ABB RAPID module: ReplayTargets_v22.mod

MODULE ReplayTargets_v22
    ! Generated from tests_v22.csv and success_v22.csv.
    ! Target names include version and testId. B* variants include version, testId, and confId.

    ! Robtargets and jointtargets for replay
    CONST robtarget rA_v22_t1 := [[2085.37,-90.629,2712.24],[0.500386,0.301254,-0.151089,0.797516],[-1,2,3,0],[9E+09,9E+09,9E+09,9E+09,9E+09,9E+09]];
    CONST robtarget rB_v22_t1 := [[2086.58,-104.628,2712.84],[0.500947,0.305697,-0.157375,0.794251],[-1,2,3,0],[9E+09,9E+09,9E+09,9E+09,9E+09,9E+09]];
    CONST robtarget rB_v22_t1_c9 := [[2086.58,-104.628,2712.84],[0.500947,0.305697,-0.157375,0.794251],[0,4,4,0],[9E+09,9E+09,9E+09,9E+09,9E+09,9E+09]];
    CONST jointtarget jA_v22_t1 := [[-0.000990208,21.9,-48.6,225.001,50.1,270.001],[9E+09,9E+09,9E+09,9E+09,9E+09,9E+09]];
    CONST jointtarget jB_v22_t1 := [[-0.330828,22.1227,-48.9906,226.207,50.1732,269.29],[9E+09,9E+09,9E+09,9E+09,9E+09,9E+09]];
    CONST jointtarget jBseed_v22_t1 := [[0,21.9,-48.6,225,50.1,270],[9E+09,9E+09,9E+09,9E+09,9E+09,9E+09]];
    CONST num seedB_v22_t1 := 12121;

    CONST robtarget rA_v22_t2 := [[2569.13,0.0397207,799.136],[0.45399,-6.87952E-6,0.891007,3.17843E-6],[0,-1,4,0],[9E+09,9E+09,9E+09,9E+09,9E+09,9E+09]];
    CONST robtarget rB_v22_t2 := [[2573.15,0.509089,797.884],[0.45376,0.0013057,0.891089,0.00778675],[0,-1,4,0],[9E+09,9E+09,9E+09,9E+09,9E+09,9E+09]];
    CONST robtarget rB_v22_t2_c8 := [[2573.15,0.509089,797.884],[0.45376,0.0013057,0.891089,0.00778675],[0,0,4,0],[9E+09,9E+09,9E+09,9E+09,9E+09,9E+09]];
    CONST jointtarget jA_v22_t2 := [[0.000888186,38.4,-6.4,-0.000518049,4,360],[9E+09,9E+09,9E+09,9E+09,9E+09,9E+09]];
    CONST jointtarget jB_v22_t2 := [[-0.0378482,38.6214,-6.68159,10.5195,4.15455,350.024],[9E+09,9E+09,9E+09,9E+09,9E+09,9E+09]];
    CONST jointtarget jBseed_v22_t2 := [[0,38.4,-6.4,0,4,360],[9E+09,9E+09,9E+09,9E+09,9E+09,9E+09]];
    CONST num seedB_v22_t2 := 701;

    CONST robtarget rA_v22_t3 := [[440.904,-79.1736,3476.31],[0.0329434,-0.13083,-0.251835,0.95832],[-1,2,3,0],[9E+09,9E+09,9E+09,9E+09,9E+09,9E+09]];
    CONST robtarget rB_v22_t3 := [[448.824,-74.9288,3477.42],[0.0397659,-0.12605,-0.257417,0.957218],[-1,2,3,0],[9E+09,9E+09,9E+09,9E+09,9E+09,9E+09]];
    CONST robtarget rB_v22_t3_c9 := [[448.824,-74.9288,3477.42],[0.0397659,-0.12605,-0.257417,0.957218],[0,4,4,0],[9E+09,9E+09,9E+09,9E+09,9E+09,9E+09]];
    CONST jointtarget jA_v22_t3 := [[-0.000733574,-1.99999,-73.1,225,42.1,315],[9E+09,9E+09,9E+09,9E+09,9E+09,9E+09]];
    CONST jointtarget jB_v22_t3 := [[0.662557,-1.16751,-74.2747,225.658,42.1266,312.818],[9E+09,9E+09,9E+09,9E+09,9E+09,9E+09]];
    CONST jointtarget jBseed_v22_t3 := [[0,-2,-73.1,225,42.1,315],[9E+09,9E+09,9E+09,9E+09,9E+09,9E+09]];
    CONST num seedB_v22_t3 := 9562;

    CONST robtarget rA_v22_t4 := [[-53.0523,1551.45,2118.27],[0.626152,-0.65099,-0.404028,-0.144592],[0,0,-2,0],[9E+09,9E+09,9E+09,9E+09,9E+09,9E+09]];
    CONST robtarget rB_v22_t4 := [[-59.1338,1553.3,2119.78],[0.622476,-0.652002,-0.408952,-0.14204],[0,0,-2,0],[9E+09,9E+09,9E+09,9E+09,9E+09,9E+09]];
    CONST robtarget rB_v22_t4_c2 := [[-59.1338,1553.3,2119.78],[0.622476,-0.652002,-0.408952,-0.14204],[0,0,-4,0],[9E+09,9E+09,9E+09,9E+09,9E+09,9E+09]];
    CONST jointtarget jA_v22_t4 := [[89.9998,-22.1,13.1,44.9995,26.7,-180],[9E+09,9E+09,9E+09,9E+09,9E+09,9E+09]];
    CONST jointtarget jB_v22_t4 := [[90.2066,-21.9258,12.8485,44.259,27.3429,-179.476],[9E+09,9E+09,9E+09,9E+09,9E+09,9E+09]];
    CONST jointtarget jBseed_v22_t4 := [[90,-22.1,13.1,45,26.7,-180],[9E+09,9E+09,9E+09,9E+09,9E+09,9E+09]];
    CONST num seedB_v22_t4 := 20938;

    CONST robtarget rA_v22_t5 := [[-90.0597,2707.57,786.857],[0.26003,0.143834,-0.650186,-0.699252],[0,-3,3,0],[9E+09,9E+09,9E+09,9E+09,9E+09,9E+09]];
    CONST robtarget rB_v22_t5 := [[-94.4005,2714.73,787.261],[0.259282,0.143229,-0.651848,-0.698106],[0,-3,3,0],[9E+09,9E+09,9E+09,9E+09,9E+09,9E+09]];
    CONST robtarget rB_v22_t5_c7 := [[-94.4005,2714.73,787.261],[0.259282,0.143229,-0.651848,-0.698106],[0,-4,4,0],[9E+09,9E+09,9E+09,9E+09,9E+09,9E+09]];
    CONST jointtarget jA_v22_t5 := [[90,47.9,-15.8,-225,49.7,315.001],[9E+09,9E+09,9E+09,9E+09,9E+09,9E+09]];
    CONST jointtarget jB_v22_t5 := [[90.1013,48.2267,-16.3618,-225.11,49.2274,315.234],[9E+09,9E+09,9E+09,9E+09,9E+09,9E+09]];
    CONST jointtarget jBseed_v22_t5 := [[90,47.9,-15.8,-225,49.7,315],[9E+09,9E+09,9E+09,9E+09,9E+09,9E+09]];
    CONST num seedB_v22_t5 := 25636;

    CONST robtarget rA_v22_t6 := [[1137.64,-69.786,3337.81],[0.705834,0.333598,0.0425546,0.623457],[-1,-2,1,0],[9E+09,9E+09,9E+09,9E+09,9E+09,9E+09]];
    CONST robtarget rB_v22_t6 := [[1136.97,-66.6338,3327.1],[0.701138,0.334311,0.0454349,0.628155],[-1,-2,1,0],[9E+09,9E+09,9E+09,9E+09,9E+09,9E+09]];
    CONST robtarget rB_v22_t6_c5 := [[1136.97,-66.6338,3327.1],[0.701138,0.334311,0.0454349,0.628155],[0,0,0,0],[9E+09,9E+09,9E+09,9E+09,9E+09,9E+09]];
    CONST jointtarget jA_v22_t6 := [[-0.000109412,5.00001,-63.4,-90.0005,24.7,179.999],[9E+09,9E+09,9E+09,9E+09,9E+09,9E+09]];
    CONST jointtarget jB_v22_t6 := [[0.115149,3.49588,-60.7888,-91.5288,24.383,182.369],[9E+09,9E+09,9E+09,9E+09,9E+09,9E+09]];
    CONST jointtarget jBseed_v22_t6 := [[0,5,-63.4,-90,24.7,180],[9E+09,9E+09,9E+09,9E+09,9E+09,9E+09]];
    CONST num seedB_v22_t6 := 26814;

    CONST robtarget rA_v22_t7 := [[-113.039,1459.37,-280.728],[0.120204,0.863598,-0.349138,-0.343296],[1,0,-2,0],[9E+09,9E+09,9E+09,9E+09,9E+09,9E+09]];
    CONST robtarget rB_v22_t7 := [[-115.209,1464.64,-290.585],[0.113531,0.8637,-0.346706,-0.347747],[1,0,-2,0],[9E+09,9E+09,9E+09,9E+09,9E+09,9E+09]];
    CONST robtarget rB_v22_t7_c2 := [[-115.209,1464.64,-290.585],[0.113531,0.8637,-0.346706,-0.347747],[0,0,-4,0],[9E+09,9E+09,9E+09,9E+09,9E+09,9E+09]];
    CONST jointtarget jA_v22_t7 := [[90,50.7,36.8,89.9993,42.6,-134.999],[9E+09,9E+09,9E+09,9E+09,9E+09,9E+09]];
    CONST jointtarget jB_v22_t7 := [[90.0686,51.3296,36.3428,91.3535,42.809,-136.629],[9E+09,9E+09,9E+09,9E+09,9E+09,9E+09]];
    CONST jointtarget jBseed_v22_t7 := [[90,50.7,36.8,90,42.6,-135],[9E+09,9E+09,9E+09,9E+09,9E+09,9E+09]];
    CONST num seedB_v22_t7 := 26900;

    CONST robtarget rA_v22_t8 := [[0.0072016,423.482,2560.63],[8.00028E-6,6.93489E-6,0.768284,0.64011],[0,-1,1,0],[9E+09,9E+09,9E+09,9E+09,9E+09,9E+09]];
    CONST robtarget rB_v22_t8 := [[8.0636,423.798,2555.65],[0.000214544,-0.00397573,-0.771793,-0.635861],[0,-1,1,0],[9E+09,9E+09,9E+09,9E+09,9E+09,9E+09]];
    CONST robtarget rB_v22_t8_c5 := [[8.0636,423.798,2555.65],[0.000214544,-0.00397573,-0.771793,-0.635861],[0,0,0,0],[9E+09,9E+09,9E+09,9E+09,9E+09,9E+09]];
    CONST jointtarget jA_v22_t8 := [[89.9992,-56.1,7.30001,-0.000484355,59.2,90.0001],[9E+09,9E+09,9E+09,9E+09,9E+09,9E+09]];
    CONST jointtarget jB_v22_t8 := [[88.3966,-56.213,7.50111,1.50836,59.7556,89.3005],[9E+09,9E+09,9E+09,9E+09,9E+09,9E+09]];
    CONST jointtarget jBseed_v22_t8 := [[90,-56.1,7.3,0,59.2,90],[9E+09,9E+09,9E+09,9E+09,9E+09,9E+09]];
    CONST num seedB_v22_t8 := 6404;

    CONST robtarget rA_v22_t9 := [[7.54404,2357.7,2259.8],[0.0143149,0.0175927,0.63119,0.775296],[1,3,2,0],[9E+09,9E+09,9E+09,9E+09,9E+09,9E+09]];
    CONST robtarget rB_v22_t9 := [[-0.0931983,2358.26,2264.28],[0.0143927,0.0137475,0.631778,0.774894],[1,3,2,0],[9E+09,9E+09,9E+09,9E+09,9E+09,9E+09]];
    CONST robtarget rB_v22_t9_c6 := [[-0.0931983,2358.26,2264.28],[0.0143927,0.0137475,0.631778,0.774894],[0,4,0,0],[9E+09,9E+09,9E+09,9E+09,9E+09,9E+09]];
    CONST jointtarget jA_v22_t9 := [[90.0008,20.9,-32.6,270,2.6,180],[9E+09,9E+09,9E+09,9E+09,9E+09,9E+09]];
    CONST jointtarget jB_v22_t9 := [[90.1746,21.034,-32.9529,276.865,2.4519,172.811],[9E+09,9E+09,9E+09,9E+09,9E+09,9E+09]];
    CONST jointtarget jBseed_v22_t9 := [[90,20.9,-32.6,270,2.6,180],[9E+09,9E+09,9E+09,9E+09,9E+09,9E+09]];
    CONST num seedB_v22_t9 := 23339;

    CONST robtarget rA_v22_t10 := [[1141.28,-1071.79,2212.75],[0.535767,-0.116814,0.733679,-0.401278],[-1,0,3,0],[9E+09,9E+09,9E+09,9E+09,9E+09,9E+09]];
    CONST robtarget rB_v22_t10 := [[1143.61,-1071.69,2219.98],[0.538493,-0.119514,0.726798,-0.409275],[-1,0,3,0],[9E+09,9E+09,9E+09,9E+09,9E+09,9E+09]];
    CONST robtarget rB_v22_t10_c8 := [[1143.61,-1071.69,2219.98],[0.538493,-0.119514,0.726798,-0.409275],[0,0,4,0],[9E+09,9E+09,9E+09,9E+09,9E+09,9E+09]];
    CONST jointtarget jA_v22_t10 := [[-45.0006,-20.3,8.59999,44.9995,24.6,270],[9E+09,9E+09,9E+09,9E+09,9E+09,9E+09]];
    CONST jointtarget jB_v22_t10 := [[-44.9215,-20.1738,8.34818,46.3284,23.7838,268.147],[9E+09,9E+09,9E+09,9E+09,9E+09,9E+09]];
    CONST jointtarget jBseed_v22_t10 := [[-45,-20.3,8.6,45,24.6,270],[9E+09,9E+09,9E+09,9E+09,9E+09,9E+09]];
    CONST num seedB_v22_t10 := 19075;

    CONST robtarget rA_v22_t11 := [[-0.0239913,-2423.41,2423.11],[0.910537,0.156457,-0.06481,0.377151],[-2,-2,3,0],[9E+09,9E+09,9E+09,9E+09,9E+09,9E+09]];
    CONST robtarget rB_v22_t11 := [[-6.2939,-2423.88,2419.9],[0.911075,0.152885,-0.070504,0.376296],[-2,-2,3,0],[9E+09,9E+09,9E+09,9E+09,9E+09,9E+09]];
    CONST robtarget rB_v22_t11_c7 := [[-6.2939,-2423.88,2419.9],[0.911075,0.152885,-0.070504,0.376296],[0,-4,4,0],[9E+09,9E+09,9E+09,9E+09,9E+09,9E+09]];
    CONST jointtarget jA_v22_t11 := [[-90.0005,35,-53.4,-180,52.1,315],[9E+09,9E+09,9E+09,9E+09,9E+09,9E+09]];
    CONST jointtarget jB_v22_t11 := [[-90.0981,34.9285,-53.1604,-179.071,52.4004,314.541],[9E+09,9E+09,9E+09,9E+09,9E+09,9E+09]];
    CONST jointtarget jBseed_v22_t11 := [[-90,35,-53.4,-180,52.1,315],[9E+09,9E+09,9E+09,9E+09,9E+09,9E+09]];
    CONST num seedB_v22_t11 := 31138;

    CONST robtarget rA_v22_t12 := [[-42.3097,-473.577,2621.44],[0.412217,-0.00327301,-0.300523,0.860089],[-1,2,-5,0],[9E+09,9E+09,9E+09,9E+09,9E+09,9E+09]];
    CONST robtarget rB_v22_t12 := [[-52.3398,-472.546,2625.75],[0.406563,-0.00528445,-0.29883,0.863354],[-1,2,-5,0],[9E+09,9E+09,9E+09,9E+09,9E+09,9E+09]];
    CONST robtarget rB_v22_t12_c2 := [[-52.3398,-472.546,2625.75],[0.406563,-0.00528445,-0.29883,0.863354],[0,0,-4,0],[9E+09,9E+09,9E+09,9E+09,9E+09,9E+09]];
    CONST jointtarget jA_v22_t12 := [[-89.999,-56.5,13.8,224.999,21,-360.001],[9E+09,9E+09,9E+09,9E+09,9E+09,9E+09]];
    CONST jointtarget jB_v22_t12 := [[-91.5149,-56.3582,13.5624,223.577,20.2415,-356.669],[9E+09,9E+09,9E+09,9E+09,9E+09,9E+09]];
    CONST jointtarget jBseed_v22_t12 := [[-90,-56.5,13.8,225,21,-360],[9E+09,9E+09,9E+09,9E+09,9E+09,9E+09]];
    CONST num seedB_v22_t12 := 22165;

    CONST robtarget rA_v22_t13 := [[-1566.34,1411.38,1591.18],[0.476074,0.481834,-0.596059,-0.431166],[1,1,-5,0],[9E+09,9E+09,9E+09,9E+09,9E+09,9E+09]];
    CONST robtarget rB_v22_t13 := [[-1558.92,1404.99,1600.09],[0.475573,0.489125,-0.596209,-0.423228],[1,1,-5,0],[9E+09,9E+09,9E+09,9E+09,9E+09,9E+09]];
    CONST robtarget rB_v22_t13_c2 := [[-1558.92,1404.99,1600.09],[0.475573,0.489125,-0.596209,-0.423228],[0,0,-4,0],[9E+09,9E+09,9E+09,9E+09,9E+09,9E+09]];
    CONST jointtarget jA_v22_t13 := [[135,5.7,7.7,90.0002,41,-360],[9E+09,9E+09,9E+09,9E+09,9E+09,9E+09]];
    CONST jointtarget jB_v22_t13 := [[134.932,5.25081,7.76172,88.089,41.843,-358.405],[9E+09,9E+09,9E+09,9E+09,9E+09,9E+09]];
    CONST jointtarget jBseed_v22_t13 := [[135,5.7,7.7,90,41,-360],[9E+09,9E+09,9E+09,9E+09,9E+09,9E+09]];
    CONST num seedB_v22_t13 := 31408;

    CONST robtarget rA_v22_t14 := [[1338.56,-1388.51,837.842],[0.215932,0.848311,-0.401491,0.269344],[-1,-1,2,0],[9E+09,9E+09,9E+09,9E+09,9E+09,9E+09]];
    CONST robtarget rB_v22_t14 := [[1345.8,-1383.01,833.682],[0.213567,0.85006,-0.393101,0.277956],[-1,-1,2,0],[9E+09,9E+09,9E+09,9E+09,9E+09,9E+09]];
    CONST robtarget rB_v22_t14_c8 := [[1345.8,-1383.01,833.682],[0.213567,0.85006,-0.393101,0.277956],[0,0,4,0],[9E+09,9E+09,9E+09,9E+09,9E+09,9E+09]];
    CONST jointtarget jA_v22_t14 := [[-45.0002,8.9,29.8,-45.001,17.4,225],[9E+09,9E+09,9E+09,9E+09,9E+09,9E+09]];
    CONST jointtarget jB_v22_t14 := [[-44.7993,9.00256,29.9162,-45.6526,16.0773,225.211],[9E+09,9E+09,9E+09,9E+09,9E+09,9E+09]];
    CONST jointtarget jBseed_v22_t14 := [[-45,8.9,29.8,-45,17.4,225],[9E+09,9E+09,9E+09,9E+09,9E+09,9E+09]];
    CONST num seedB_v22_t14 := 14462;

    CONST robtarget rA_v22_t15 := [[1463.5,1463.45,-50.4844],[1.32519E-6,-0.703743,-0.703721,0.0975829],[0,0,-3,0],[9E+09,9E+09,9E+09,9E+09,9E+09,9E+09]];
    CONST robtarget rB_v22_t15 := [[1464.94,1453.65,-55.8845],[0.0062937,0.70434,0.703424,-0.0951863],[0,0,-3,0],[9E+09,9E+09,9E+09,9E+09,9E+09,9E+09]];
    CONST robtarget rB_v22_t15_c2 := [[1464.94,1453.65,-55.8845],[0.0062937,0.70434,0.703424,-0.0951863],[0,0,-4,0],[9E+09,9E+09,9E+09,9E+09,9E+09,9E+09]];
    CONST jointtarget jA_v22_t15 := [[44.9991,50.8,10.7,0.000226803,39.7,-224.999],[9E+09,9E+09,9E+09,9E+09,9E+09,9E+09]];
    CONST jointtarget jB_v22_t15 := [[44.8383,50.8187,10.9944,-1.1754,39.116,-224.104],[9E+09,9E+09,9E+09,9E+09,9E+09,9E+09]];
    CONST jointtarget jBseed_v22_t15 := [[45,50.8,10.7,0,39.7,-225],[9E+09,9E+09,9E+09,9E+09,9E+09,9E+09]];
    CONST num seedB_v22_t15 := 29029;

    CONST robtarget rA_v22_t16 := [[-1120.18,-991.21,1224.1],[0.422333,-0.451194,-0.676806,0.39999],[-2,-1,-4,0],[9E+09,9E+09,9E+09,9E+09,9E+09,9E+09]];
    CONST robtarget rB_v22_t16 := [[-1118.1,-991.976,1220.42],[0.419661,-0.446818,-0.67964,0.402899],[-2,-1,-4,0],[9E+09,9E+09,9E+09,9E+09,9E+09,9E+09]];
    CONST robtarget rB_v22_t16_c2 := [[-1118.1,-991.976,1220.42],[0.419661,-0.446818,-0.67964,0.402899],[0,0,-4,0],[9E+09,9E+09,9E+09,9E+09,9E+09,9E+09]];
    CONST jointtarget jA_v22_t16 := [[-135,-24.3,47,-89.9996,33.1,-359.999],[9E+09,9E+09,9E+09,9E+09,9E+09,9E+09]];
    CONST jointtarget jB_v22_t16 := [[-134.987,-24.371,47.1904,-90.496,32.4172,-359.736],[9E+09,9E+09,9E+09,9E+09,9E+09,9E+09]];
    CONST jointtarget jBseed_v22_t16 := [[-135,-24.3,47,-90,33.1,-360],[9E+09,9E+09,9E+09,9E+09,9E+09,9E+09]];
    CONST num seedB_v22_t16 := 29294;

    CONST robtarget rA_v22_t17 := [[-1678.82,1673.45,2048.89],[0.00774962,0.488526,-0.476806,-0.730711],[1,-4,3,0],[9E+09,9E+09,9E+09,9E+09,9E+09,9E+09]];
    CONST robtarget rB_v22_t17 := [[-1684.57,1677.08,2047.65],[0.0130046,0.48471,-0.480159,-0.730982],[1,-4,3,0],[9E+09,9E+09,9E+09,9E+09,9E+09,9E+09]];
    CONST robtarget rB_v22_t17_c7 := [[-1684.57,1677.08,2047.65],[0.0130046,0.48471,-0.480159,-0.730982],[0,-4,4,0],[9E+09,9E+09,9E+09,9E+09,9E+09,9E+09]];
    CONST jointtarget jA_v22_t17 := [[135,18.4,-22.3,-270,1.3,315.001],[9E+09,9E+09,9E+09,9E+09,9E+09,9E+09]];
    CONST jointtarget jB_v22_t17 := [[135.04,18.768,-22.7011,-268.86,1.24664,314.695],[9E+09,9E+09,9E+09,9E+09,9E+09,9E+09]];
    CONST jointtarget jBseed_v22_t17 := [[135,18.4,-22.3,-270,1.3,315],[9E+09,9E+09,9E+09,9E+09,9E+09,9E+09]];
    CONST num seedB_v22_t17 := 13883;

    CONST robtarget rA_v22_t19 := [[1387.04,1386.99,2336.67],[0.49031,-0.720551,1.06996E-5,-0.490308],[0,0,2,0],[9E+09,9E+09,9E+09,9E+09,9E+09,9E+09]];
    CONST robtarget rB_v22_t19 := [[1387.99,1390.13,2325.49],[0.487063,-0.718691,0.00617927,-0.496199],[0,0,2,0],[9E+09,9E+09,9E+09,9E+09,9E+09,9E+09]];
    CONST robtarget rB_v22_t19_c8 := [[1387.99,1390.13,2325.49],[0.487063,-0.718691,0.00617927,-0.496199],[0,0,4,0],[9E+09,9E+09,9E+09,9E+09,9E+09,9E+09]];
    CONST jointtarget jA_v22_t19 := [[44.9991,0.800001,-14.2,0.000667401,15.6,225],[9E+09,9E+09,9E+09,9E+09,9E+09,9E+09]];
    CONST jointtarget jB_v22_t19 := [[45.1433,0.716712,-13.6432,-4.5546,14.8692,229.402],[9E+09,9E+09,9E+09,9E+09,9E+09,9E+09]];
    CONST jointtarget jBseed_v22_t19 := [[45,0.8,-14.2,0,15.6,225],[9E+09,9E+09,9E+09,9E+09,9E+09,9E+09]];
    CONST num seedB_v22_t19 := 19067;

    CONST robtarget rA_v22_t20 := [[-80.2355,-213.269,2838.92],[0.824752,0.503204,-0.248139,-0.0706906],[-2,-1,-3,0],[9E+09,9E+09,9E+09,9E+09,9E+09,9E+09]];
    CONST robtarget rB_v22_t20 := [[-83.549,-218.941,2831.62],[0.825653,0.500928,-0.251418,-0.064484],[-2,-1,-3,0],[9E+09,9E+09,9E+09,9E+09,9E+09,9E+09]];
    CONST robtarget rB_v22_t20_c2 := [[-83.549,-218.941,2831.62],[0.825653,0.500928,-0.251418,-0.064484],[0,0,-4,0],[9E+09,9E+09,9E+09,9E+09,9E+09,9E+09]];
    CONST jointtarget jA_v22_t20 := [[-90.0003,-52.2,-6,-45.0009,42.8,-225],[9E+09,9E+09,9E+09,9E+09,9E+09,9E+09]];
    CONST jointtarget jB_v22_t20 := [[-92.2764,-52.4324,-5.4223,-42.3815,41.6336,-225.087],[9E+09,9E+09,9E+09,9E+09,9E+09,9E+09]];
    CONST jointtarget jBseed_v22_t20 := [[-90,-52.2,-6,-45,42.8,-225],[9E+09,9E+09,9E+09,9E+09,9E+09,9E+09]];
    CONST num seedB_v22_t20 := 16887;

    CONST robtarget rA_v22_t21 := [[-923.186,923.189,1598.86],[0.604509,-0.518773,7.16223E-6,0.604519],[1,2,1,0],[9E+09,9E+09,9E+09,9E+09,9E+09,9E+09]];
    CONST robtarget rB_v22_t21 := [[-931.406,926.916,1600.61],[0.610799,-0.51017,-0.0036644,0.605506],[1,2,1,0],[9E+09,9E+09,9E+09,9E+09,9E+09,9E+09]];
    CONST robtarget rB_v22_t21_c5 := [[-931.406,926.916,1600.61],[0.610799,-0.51017,-0.0036644,0.605506],[0,0,0,0],[9E+09,9E+09,9E+09,9E+09,9E+09,9E+09]];
    CONST jointtarget jA_v22_t21 := [[135,-40.2,47.7,180,35,135.001],[9E+09,9E+09,9E+09,9E+09,9E+09,9E+09]];
    CONST jointtarget jB_v22_t21 := [[135.135,-39.5283,47.3815,179.961,36.5011,134.384],[9E+09,9E+09,9E+09,9E+09,9E+09,9E+09]];
    CONST jointtarget jBseed_v22_t21 := [[135,-40.2,47.7,180,35,135],[9E+09,9E+09,9E+09,9E+09,9E+09,9E+09]];
    CONST num seedB_v22_t21 := 26637;

    CONST robtarget rA_v22_t22 := [[950.54,-840.515,1691.42],[0.0297644,0.836296,-0.153509,0.525507],[-1,0,-3,0],[9E+09,9E+09,9E+09,9E+09,9E+09,9E+09]];
    CONST robtarget rB_v22_t22 := [[960.745,-837.04,1696.54],[0.0318737,0.839278,-0.149814,0.521683],[-1,0,-3,0],[9E+09,9E+09,9E+09,9E+09,9E+09,9E+09]];
    CONST robtarget rB_v22_t22_c2 := [[960.745,-837.04,1696.54],[0.0318737,0.839278,-0.149814,0.521683],[0,0,-4,0],[9E+09,9E+09,9E+09,9E+09,9E+09,9E+09]];
    CONST jointtarget jA_v22_t22 := [[-44.9992,-40.2,38.7,44.9993,41.2,-224.999],[9E+09,9E+09,9E+09,9E+09,9E+09,9E+09]];
    CONST jointtarget jB_v22_t22 := [[-44.5007,-39.8223,38.2603,43.9606,41.2216,-224.512],[9E+09,9E+09,9E+09,9E+09,9E+09,9E+09]];
    CONST jointtarget jBseed_v22_t22 := [[-45,-40.2,38.7,45,41.2,-225],[9E+09,9E+09,9E+09,9E+09,9E+09,9E+09]];
    CONST num seedB_v22_t22 := 21583;

    CONST robtarget rA_v22_t23 := [[1958.85,-1802.66,2190.57],[0.687421,-0.292183,0.526473,-0.406088],[-1,0,-2,0],[9E+09,9E+09,9E+09,9E+09,9E+09,9E+09]];
    CONST robtarget rB_v22_t23 := [[1954.37,-1806.34,2193.79],[0.683778,-0.293726,0.530505,-0.405879],[-1,0,-2,0],[9E+09,9E+09,9E+09,9E+09,9E+09,9E+09]];
    CONST robtarget rB_v22_t23_c5 := [[1954.37,-1806.34,2193.79],[0.683778,-0.293726,0.530505,-0.405879],[0,0,0,0],[9E+09,9E+09,9E+09,9E+09,9E+09,9E+09]];
    CONST jointtarget jA_v22_t23 := [[-44.9999,49.9,-71.4,89.9994,41.4,-135],[9E+09,9E+09,9E+09,9E+09,9E+09,9E+09]];
    CONST jointtarget jB_v22_t23 := [[-45.1292,50.2553,-72.1866,88.5969,41.5219,-133.74],[9E+09,9E+09,9E+09,9E+09,9E+09,9E+09]];
    CONST jointtarget jBseed_v22_t23 := [[-45,49.9,-71.4,90,41.4,-135],[9E+09,9E+09,9E+09,9E+09,9E+09,9E+09]];
    CONST num seedB_v22_t23 := 10285;

    CONST robtarget rA_v22_t24 := [[1909.05,-45.5577,779.791],[0.309343,0.416833,0.854681,-0.008768],[0,-1,1,0],[9E+09,9E+09,9E+09,9E+09,9E+09,9E+09]];
    CONST robtarget rB_v22_t24 := [[1902.13,-47.5464,775.692],[0.312787,0.424986,0.849344,-0.0128888],[0,-1,1,0],[9E+09,9E+09,9E+09,9E+09,9E+09,9E+09]];
    CONST robtarget rB_v22_t24_c2 := [[1902.13,-47.5464,775.692],[0.312787,0.424986,0.849344,-0.0128888],[0,0,-4,0],[9E+09,9E+09,9E+09,9E+09,9E+09,9E+09]];
    CONST robtarget rB_v22_t24_c5 := [[1902.13,-47.5464,775.692],[0.312787,0.424986,0.849344,-0.0128888],[0,0,0,0],[9E+09,9E+09,9E+09,9E+09,9E+09,9E+09]];
    CONST jointtarget jA_v22_t24 := [[0.000398436,10.2,30.5,-45.0007,22.7,90],[9E+09,9E+09,9E+09,9E+09,9E+09,9E+09]];
    CONST jointtarget jB_v22_t24 := [[0.0160526,10.0353,30.9027,-47.2174,23.0957,93.0322],[9E+09,9E+09,9E+09,9E+09,9E+09,9E+09]];
    CONST jointtarget jBseed_v22_t24 := [[0,10.2,30.5,-45,22.7,90],[9E+09,9E+09,9E+09,9E+09,9E+09,9E+09]];
    CONST num seedB_v22_t24 := 28996;

    CONST robtarget rA_v22_t25 := [[-1491.49,1435.7,2615.86],[0.57706,-0.453381,-0.099156,0.672023],[1,1,-2,0],[9E+09,9E+09,9E+09,9E+09,9E+09,9E+09]];
    CONST robtarget rB_v22_t25 := [[-1498.42,1440.53,2607.51],[0.577707,-0.457317,-0.0961145,0.669237],[1,1,-2,0],[9E+09,9E+09,9E+09,9E+09,9E+09,9E+09]];
    CONST robtarget rB_v22_t25_c2 := [[-1498.42,1440.53,2607.51],[0.577707,-0.457317,-0.0961145,0.669237],[0,0,-4,0],[9E+09,9E+09,9E+09,9E+09,9E+09,9E+09]];
    CONST jointtarget jA_v22_t25 := [[135.001,13.2,-35,135.001,19.5,-180],[9E+09,9E+09,9E+09,9E+09,9E+09,9E+09]];
    CONST jointtarget jB_v22_t25 := [[135.081,13.3914,-34.919,135.611,18.9849,-180.715],[9E+09,9E+09,9E+09,9E+09,9E+09,9E+09]];
    CONST jointtarget jBseed_v22_t25 := [[135,13.2,-35,135,19.5,-180],[9E+09,9E+09,9E+09,9E+09,9E+09,9E+09]];
    CONST num seedB_v22_t25 := 28430;

    CONST robtarget rA_v22_t26 := [[-1362.76,-1300.42,-378.575],[0.16703,-0.391188,-0.903177,0.0578325],[-2,-1,0,0],[9E+09,9E+09,9E+09,9E+09,9E+09,9E+09]];
    CONST robtarget rB_v22_t26 := [[-1357.88,-1299.28,-389.537],[0.176509,-0.391477,-0.901208,0.0584293],[-2,-1,0,0],[9E+09,9E+09,9E+09,9E+09,9E+09,9E+09]];
    CONST robtarget rB_v22_t26_c5 := [[-1357.88,-1299.28,-389.537],[0.176509,-0.391477,-0.901208,0.0584293],[0,0,0,0],[9E+09,9E+09,9E+09,9E+09,9E+09,9E+09]];
    CONST jointtarget jA_v22_t26 := [[-135.001,59.7,16.7,-89.9993,15.3,0.000855239],[9E+09,9E+09,9E+09,9E+09,9E+09,9E+09]];
    CONST jointtarget jB_v22_t26 := [[-134.831,60.1848,16.6162,-92.9555,16.3571,3.17921],[9E+09,9E+09,9E+09,9E+09,9E+09,9E+09]];
    CONST jointtarget jBseed_v22_t26 := [[-135,59.7,16.7,-90,15.3,0],[9E+09,9E+09,9E+09,9E+09,9E+09,9E+09]];
    CONST num seedB_v22_t26 := 15153;

    CONST robtarget rA_v22_t27 := [[1130.17,1166.91,1200.62],[0.595087,-0.595016,0.536137,0.0662089],[0,1,1,0],[9E+09,9E+09,9E+09,9E+09,9E+09,9E+09]];
    CONST robtarget rB_v22_t27 := [[1132.56,1154.11,1205.03],[0.602094,-0.586605,0.536689,0.0730895],[0,1,1,0],[9E+09,9E+09,9E+09,9E+09,9E+09,9E+09]];
    CONST robtarget rB_v22_t27_c4 := [[1132.56,1154.11,1205.03],[0.602094,-0.586605,0.536689,0.0730895],[0,-4,0,0],[9E+09,9E+09,9E+09,9E+09,9E+09,9E+09]];
    CONST robtarget rB_v22_t27_c5 := [[1132.56,1154.11,1205.03],[0.602094,-0.586605,0.536689,0.0730895],[0,0,0,0],[9E+09,9E+09,9E+09,9E+09,9E+09,9E+09]];
    CONST jointtarget jA_v22_t27 := [[45.0005,-17.4,43.1,134.999,12.7,179.999],[9E+09,9E+09,9E+09,9E+09,9E+09,9E+09]];
    CONST jointtarget jB_v22_t27 := [[44.5578,-17.913,43.4458,135.864,13.7866,180.033],[9E+09,9E+09,9E+09,9E+09,9E+09,9E+09]];
    CONST jointtarget jBseed_v22_t27 := [[45,-17.4,43.1,135,12.7,180],[9E+09,9E+09,9E+09,9E+09,9E+09,9E+09]];
    CONST num seedB_v22_t27 := 361;

    CONST robtarget rA_v22_t28 := [[-412.494,412.501,3202.83],[0.999086,0.0302279,0.0302262,-9.08665E-6],[1,-3,0,0],[9E+09,9E+09,9E+09,9E+09,9E+09,9E+09]];
    CONST robtarget rB_v22_t28 := [[-417.962,410.543,3199.39],[0.99898,0.0243203,0.037032,0.00869105],[1,-3,0,0],[9E+09,9E+09,9E+09,9E+09,9E+09,9E+09]];
    CONST robtarget rB_v22_t28_c4 := [[-417.962,410.543,3199.39],[0.99898,0.0243203,0.037032,0.00869105],[0,-4,0,0],[9E+09,9E+09,9E+09,9E+09,9E+09,9E+09]];
    CONST jointtarget jA_v22_t28 := [[134.999,-25.9,-27.3,-180,41.7,44.9996],[9E+09,9E+09,9E+09,9E+09,9E+09,9E+09]];
    CONST jointtarget jB_v22_t28 := [[135.799,-25.9999,-27.011,-178.5,41.9776,44.0393],[9E+09,9E+09,9E+09,9E+09,9E+09,9E+09]];
    CONST jointtarget jBseed_v22_t28 := [[135,-25.9,-27.3,-180,41.7,45],[9E+09,9E+09,9E+09,9E+09,9E+09,9E+09]];
    CONST num seedB_v22_t28 := 14096;

    CONST robtarget rA_v22_t29 := [[1491.94,65.5074,3240.43],[0.974161,-0.195319,0.0948671,0.0621398],[-1,1,-2,0],[9E+09,9E+09,9E+09,9E+09,9E+09,9E+09]];
    CONST robtarget rB_v22_t29 := [[1487.65,62.1208,3242.65],[0.973589,-0.197748,0.0958919,0.0618472],[-1,1,-2,0],[9E+09,9E+09,9E+09,9E+09,9E+09,9E+09]];
    CONST robtarget rB_v22_t29_c5 := [[1487.65,62.1208,3242.65],[0.973589,-0.197748,0.0958919,0.0618472],[0,0,0,0],[9E+09,9E+09,9E+09,9E+09,9E+09,9E+09]];
    CONST jointtarget jA_v22_t29 := [[-0.000492133,21.7,-76.4,135,33.7,-135],[9E+09,9E+09,9E+09,9E+09,9E+09,9E+09]];
    CONST jointtarget jB_v22_t29 := [[-0.163329,21.7881,-76.7439,134.229,33.6806,-134.143],[9E+09,9E+09,9E+09,9E+09,9E+09,9E+09]];
    CONST jointtarget jBseed_v22_t29 := [[0,21.7,-76.4,135,33.7,-135],[9E+09,9E+09,9E+09,9E+09,9E+09,9E+09]];
    CONST num seedB_v22_t29 := 29740;

    CONST robtarget rA_v22_t30 := [[103.299,-2100.89,322.216],[0.179201,-0.435941,0.794624,-0.382642],[-1,-3,-3,0],[9E+09,9E+09,9E+09,9E+09,9E+09,9E+09]];
    CONST robtarget rB_v22_t30 := [[96.8713,-2104.95,316.793],[0.174169,-0.434041,0.797979,-0.380136],[-1,-3,-3,0],[9E+09,9E+09,9E+09,9E+09,9E+09,9E+09]];
    CONST robtarget rB_v22_t30_c1 := [[96.8713,-2104.95,316.793],[0.174169,-0.434041,0.797979,-0.380136],[0,-4,-4,0],[9E+09,9E+09,9E+09,9E+09,9E+09,9E+09]];
    CONST jointtarget jA_v22_t30 := [[-89.9993,35.6,19.3,-269.999,38.2,-225],[9E+09,9E+09,9E+09,9E+09,9E+09,9E+09]];
    CONST jointtarget jB_v22_t30 := [[-90.1315,35.8838,19.0678,-270.161,37.5173,-224.818],[9E+09,9E+09,9E+09,9E+09,9E+09,9E+09]];
    CONST jointtarget jBseed_v22_t30 := [[-90,35.6,19.3,-270,38.2,-225],[9E+09,9E+09,9E+09,9E+09,9E+09,9E+09]];
    CONST num seedB_v22_t30 := 29168;

    CONST robtarget rA_v22_t31 := [[-129.2,2085.24,276.271],[0.258184,-0.866046,-0.122313,0.4103],[0,-4,1,0],[9E+09,9E+09,9E+09,9E+09,9E+09,9E+09]];
    CONST robtarget rB_v22_t31 := [[-131.972,2080.28,283.701],[0.259111,-0.865404,-0.130757,0.408462],[0,-4,1,0],[9E+09,9E+09,9E+09,9E+09,9E+09,9E+09]];
    CONST robtarget rB_v22_t31_c4 := [[-131.972,2080.28,283.701],[0.259111,-0.865404,-0.130757,0.408462],[0,-4,0,0],[9E+09,9E+09,9E+09,9E+09,9E+09,9E+09]];
    CONST jointtarget jA_v22_t31 := [[89.9991,38.2,18.6,-270,50.7,180],[9E+09,9E+09,9E+09,9E+09,9E+09,9E+09]];
    CONST jointtarget jB_v22_t31 := [[90.0734,37.7528,18.9122,-270.452,50.743,179.484],[9E+09,9E+09,9E+09,9E+09,9E+09,9E+09]];
    CONST jointtarget jBseed_v22_t31 := [[90,38.2,18.6,-270,50.7,180],[9E+09,9E+09,9E+09,9E+09,9E+09,9E+09]];
    CONST num seedB_v22_t31 := 26505;

    CONST robtarget rA_v22_t32 := [[-98.3785,-1309.86,2900.82],[0.546614,0.299267,-0.115237,-0.773546],[-2,-2,-3,0],[9E+09,9E+09,9E+09,9E+09,9E+09,9E+09]];
    CONST robtarget rB_v22_t32 := [[-93.119,-1304.73,2909.86],[0.548838,0.303153,-0.107306,-0.771596],[-2,-2,-3,0],[9E+09,9E+09,9E+09,9E+09,9E+09,9E+09]];
    CONST robtarget rB_v22_t32_c2 := [[-93.119,-1304.73,2909.86],[0.548838,0.303153,-0.107306,-0.771596],[0,0,-4,0],[9E+09,9E+09,9E+09,9E+09,9E+09,9E+09]];
    CONST jointtarget jA_v22_t32 := [[-90.0009,-11.9,-20.7,-134.999,56.4,-225],[9E+09,9E+09,9E+09,9E+09,9E+09,9E+09]];
    CONST jointtarget jB_v22_t32 := [[-89.7901,-11.9164,-21.1306,-134.44,55.1896,-225.748],[9E+09,9E+09,9E+09,9E+09,9E+09,9E+09]];
    CONST jointtarget jBseed_v22_t32 := [[-90,-11.9,-20.7,-135,56.4,-225],[9E+09,9E+09,9E+09,9E+09,9E+09,9E+09]];
    CONST num seedB_v22_t32 := 4165;

    CONST robtarget rA_v22_t34 := [[-13.142,-1283.57,2012.29],[0.535253,0.460383,0.418066,-0.57164],[-1,-2,-3,0],[9E+09,9E+09,9E+09,9E+09,9E+09,9E+09]];
    CONST robtarget rB_v22_t34 := [[-6.42479,-1285.41,2002.95],[0.527772,0.461212,0.417196,-0.578522],[-1,-2,-3,0],[9E+09,9E+09,9E+09,9E+09,9E+09,9E+09]];
    CONST robtarget rB_v22_t34_c2 := [[-6.42479,-1285.41,2002.95],[0.527772,0.461212,0.417196,-0.578522],[0,0,-4,0],[9E+09,9E+09,9E+09,9E+09,9E+09,9E+09]];
    CONST robtarget rB_v22_t34_c5 := [[-6.42479,-1285.41,2002.95],[0.527772,0.461212,0.417196,-0.578522],[0,0,0,0],[9E+09,9E+09,9E+09,9E+09,9E+09,9E+09]];
    CONST jointtarget jA_v22_t34 := [[-89.9991,-38.6,30,-134.999,6.4,-225],[9E+09,9E+09,9E+09,9E+09,9E+09,9E+09]];
    CONST jointtarget jB_v22_t34 := [[-89.5333,-38.6294,30.3716,-130.029,7.59213,-230.835],[9E+09,9E+09,9E+09,9E+09,9E+09,9E+09]];
    CONST jointtarget jBseed_v22_t34 := [[-90,-38.6,30,-135,6.4,-225],[9E+09,9E+09,9E+09,9E+09,9E+09,9E+09]];
    CONST num seedB_v22_t34 := 25608;

    CONST robtarget rA_v22_t35 := [[-1536.97,1652.77,1643.97],[0.642333,-0.367391,-0.459845,-0.490892],[1,2,3,0],[9E+09,9E+09,9E+09,9E+09,9E+09,9E+09]];
    CONST robtarget rB_v22_t35 := [[-1541.44,1650.53,1644.05],[0.647258,-0.369347,-0.454738,-0.487702],[1,2,3,0],[9E+09,9E+09,9E+09,9E+09,9E+09,9E+09]];
    CONST robtarget rB_v22_t35_c5 := [[-1541.44,1650.53,1644.05],[0.647258,-0.369347,-0.454738,-0.487702],[0,0,0,0],[9E+09,9E+09,9E+09,9E+09,9E+09,9E+09]];
    CONST robtarget rB_v22_t35_c8 := [[-1541.44,1650.53,1644.05],[0.647258,-0.369347,-0.454738,-0.487702],[0,0,4,0],[9E+09,9E+09,9E+09,9E+09,9E+09,9E+09]];
    CONST jointtarget jA_v22_t35 := [[135,12.8,0.800005,225,43.9,315],[9E+09,9E+09,9E+09,9E+09,9E+09,9E+09]];
    CONST jointtarget jB_v22_t35 := [[135.128,12.907,0.712501,224.769,44.3193,315.965],[9E+09,9E+09,9E+09,9E+09,9E+09,9E+09]];
    CONST jointtarget jBseed_v22_t35 := [[135,12.8,0.8,225,43.9,315],[9E+09,9E+09,9E+09,9E+09,9E+09,9E+09]];
    CONST num seedB_v22_t35 := 7511;

ENDMODULE
